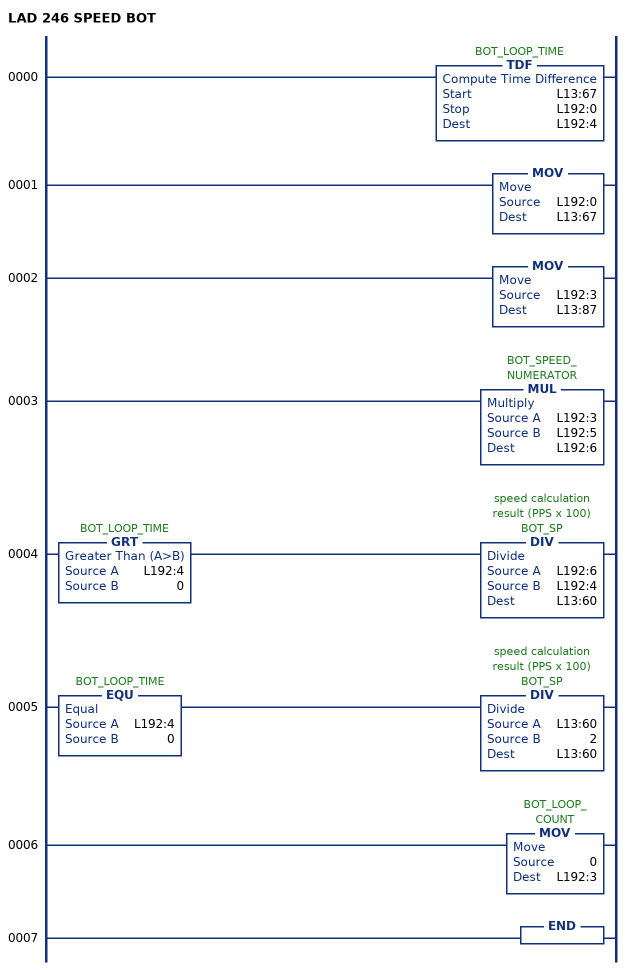
% Rung: 0 %
SOR TDF L13:67 L192:0 L192:4 EOR
%   L192:0  BOT_THIS_TIME  "rtc bot belt movement event time" %
%   L192:4  BOT_LOOP_TIME %
% Rung: 1 %
SOR MOV L192:0 L13:67 EOR
%   L192:0  BOT_THIS_TIME  "rtc bot belt movement event time" %
% Rung: 2 %
SOR MOV L192:3 L13:87 EOR
%   L192:3  BOT_LOOP_COUNT %
% Rung: 3 %
SOR MUL L192:3 L192:5 L192:6 EOR
%   L192:3  BOT_LOOP_COUNT %
%   L192:5  TKS_PER_SECOND %
%   L192:6  BOT_SPEED_NUMERATOR %
% Rung: 4 %
SOR GRT L192:4 0 DIV L192:6 L192:4 L13:60 EOR
%   L192:4  BOT_LOOP_TIME %
%   L192:6  BOT_SPEED_NUMERATOR %
%   L13:60  BOT_SP  "speed calculation result (PPS x 100)" %
% Rung: 5 %
SOR EQU L192:4 0 DIV L13:60 2 L13:60 EOR
%   L192:4  BOT_LOOP_TIME %
%   L13:60  BOT_SP  "speed calculation result (PPS x 100)" %
% Rung: 6 %
SOR MOV 0 L192:3 EOR
%   L192:3  BOT_LOOP_COUNT %
% Rung: 7 %
SOR END EOR

LADDER 248 "SPEED TOP"    % high speed %
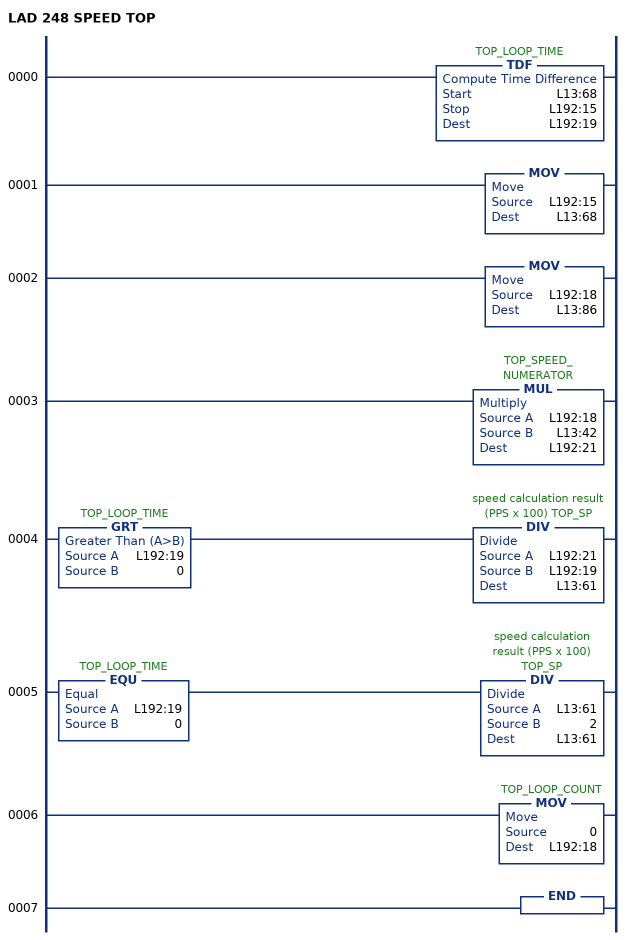
% Rung: 0 %
SOR TDF L13:68 L192:15 L192:19 EOR
%   L192:15  TOP_THIS_TIME  "rtc top belt movement event time" %
%   L192:19  TOP_LOOP_TIME %
% Rung: 1 %
SOR MOV L192:15 L13:68 EOR
%   L192:15  TOP_THIS_TIME  "rtc top belt movement event time" %
% Rung: 2 %
SOR MOV L192:18 L13:86 EOR
%   L192:18  TOP_LOOP_COUNT %
% Rung: 3 %
SOR MUL L192:18 L13:42 L192:21 EOR
%   L192:18  TOP_LOOP_COUNT %
%   L192:21  TOP_SPEED_NUMERATOR %
% Rung: 4 %
SOR GRT L192:19 0 DIV L192:21 L192:19 L13:61 EOR
%   L192:19  TOP_LOOP_TIME %
%   L192:21  TOP_SPEED_NUMERATOR %
%   L13:61  TOP_SP  "speed calculation result (PPS x 100)" %
% Rung: 5 %
SOR EQU L192:19 0 DIV L13:61 2 L13:61 EOR
%   L192:19  TOP_LOOP_TIME %
%   L13:61  TOP_SP  "speed calculation result (PPS x 100)" %
% Rung: 6 %
SOR MOV 0 L192:18 EOR
%   L192:18  TOP_LOOP_COUNT %
% Rung: 7 %
SOR END EOR

LADDER 250 "P BOT"    % high speed %
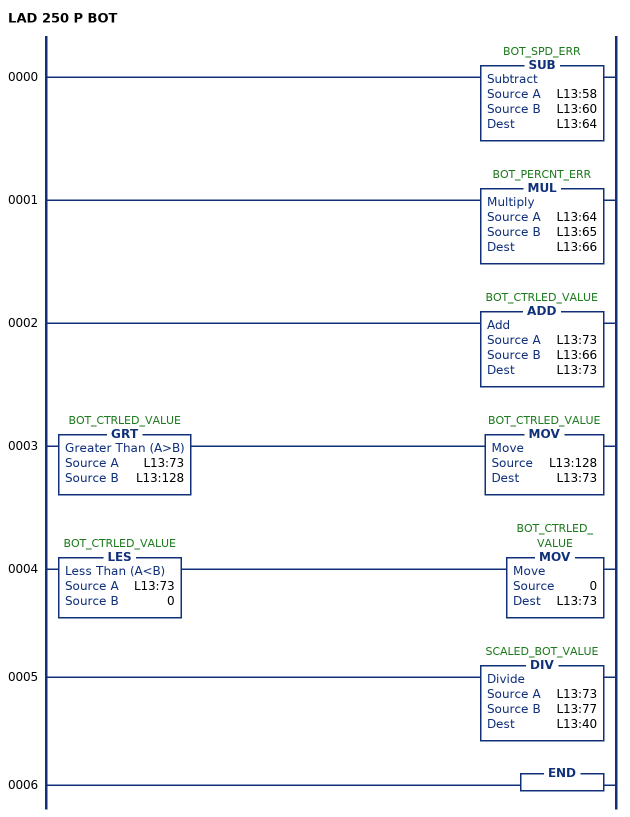
% Rung: 0 %
SOR SUB L13:58 L13:60 L13:64 EOR
%   L13:58  BOT_SPD_SETPOINT %
%   L13:60  BOT_SP  "speed calculation result (PPS x 100)" %
%   L13:64  BOT_SPD_ERR %
% Rung: 1 %
SOR MUL L13:64 L13:65 L13:66 EOR
%   L13:64  BOT_SPD_ERR %
%   L13:65  POS5SHIFT %
%   L13:66  BOT_PERCNT_ERR %
% Rung: 2 %
SOR ADD L13:73 L13:66 L13:73 EOR
%   L13:73  BOT_CTRLED_VALUE %
%   L13:66  BOT_PERCNT_ERR %
% Rung: 3 %
SOR GRT L13:73 L13:128 MOV L13:128 L13:73 EOR
%   L13:73  BOT_CTRLED_VALUE %
%   L13:128  "how much top has shifted since measurment" %
% Rung: 4 %
SOR LES L13:73 0 MOV 0 L13:73 EOR
%   L13:73  BOT_CTRLED_VALUE %
% Rung: 5 %
SOR DIV L13:73 L13:77 L13:40 EOR
%   L13:73  BOT_CTRLED_VALUE %
%   L13:40  SCALED_BOT_VALUE %
% Rung: 6 %
SOR END EOR

LADDER 252 "P TOP"    % high speed %
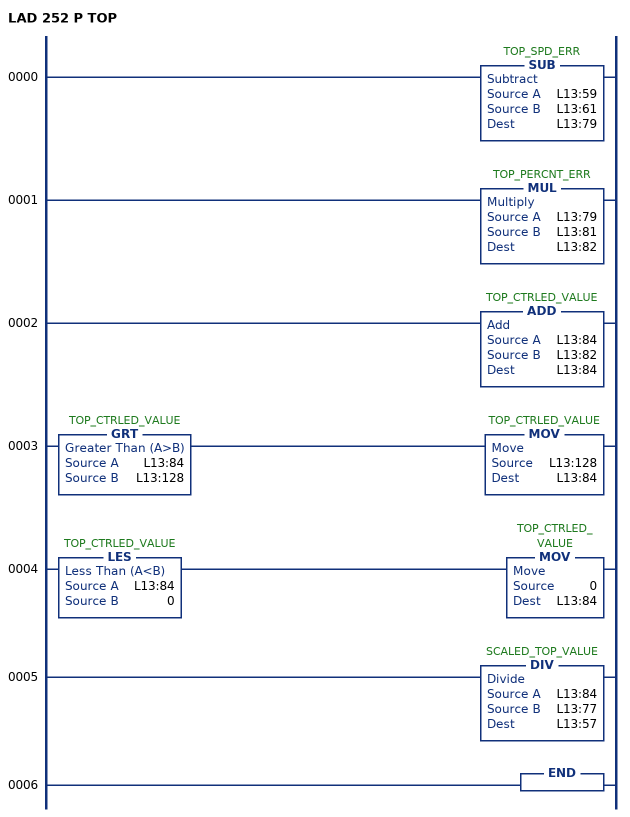
% Rung: 0 %
SOR SUB L13:59 L13:61 L13:79 EOR
%   L13:59  TOP_SPD_SETPOINT %
%   L13:61  TOP_SP  "speed calculation result (PPS x 100)" %
%   L13:79  TOP_SPD_ERR %
% Rung: 1 %
SOR MUL L13:79 L13:81 L13:82 EOR
%   L13:79  TOP_SPD_ERR %
%   L13:81  TOP_FDBK_RATIO %
%   L13:82  TOP_PERCNT_ERR %
% Rung: 2 %
SOR ADD L13:84 L13:82 L13:84 EOR
%   L13:84  TOP_CTRLED_VALUE %
%   L13:82  TOP_PERCNT_ERR %
% Rung: 3 %
SOR GRT L13:84 L13:128 MOV L13:128 L13:84 EOR
%   L13:84  TOP_CTRLED_VALUE %
%   L13:128  "how much top has shifted since measurment" %
% Rung: 4 %
SOR LES L13:84 0 MOV 0 L13:84 EOR
%   L13:84  TOP_CTRLED_VALUE %
% Rung: 5 %
SOR DIV L13:84 L13:77 L13:57 EOR
%   L13:84  TOP_CTRLED_VALUE %
%   L13:57  SCALED_TOP_VALUE %
% Rung: 6 %
SOR END EOR

LADDER 254 "TOTALCOUNT"
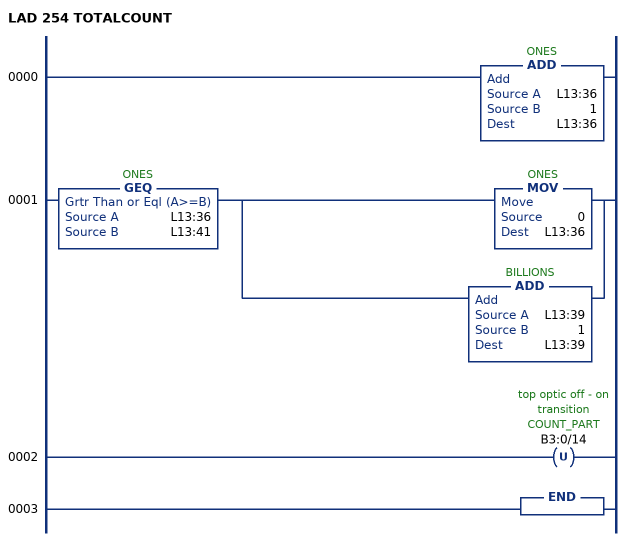
% Rung: 0 %
SOR ADD L13:36 1 L13:36 EOR
%   L13:36  ONES %
% Rung: 1 %
SOR GEQ L13:36 L13:41 BST MOV 0 L13:36 NXB ADD L13:39 1 L13:39 BND EOR
%   L13:36  ONES %
%   L13:41  "skipped count change in the last 3 seconds" %
%   L13:39  BILLIONS %
% Rung: 2 %
SOR OTU B3:0/14 EOR
%   B3:0/14  COUNT_PART  "top optic off - on transition" %
% Rung: 3 %
SOR END EOR

LADDER 255 "SAVED"
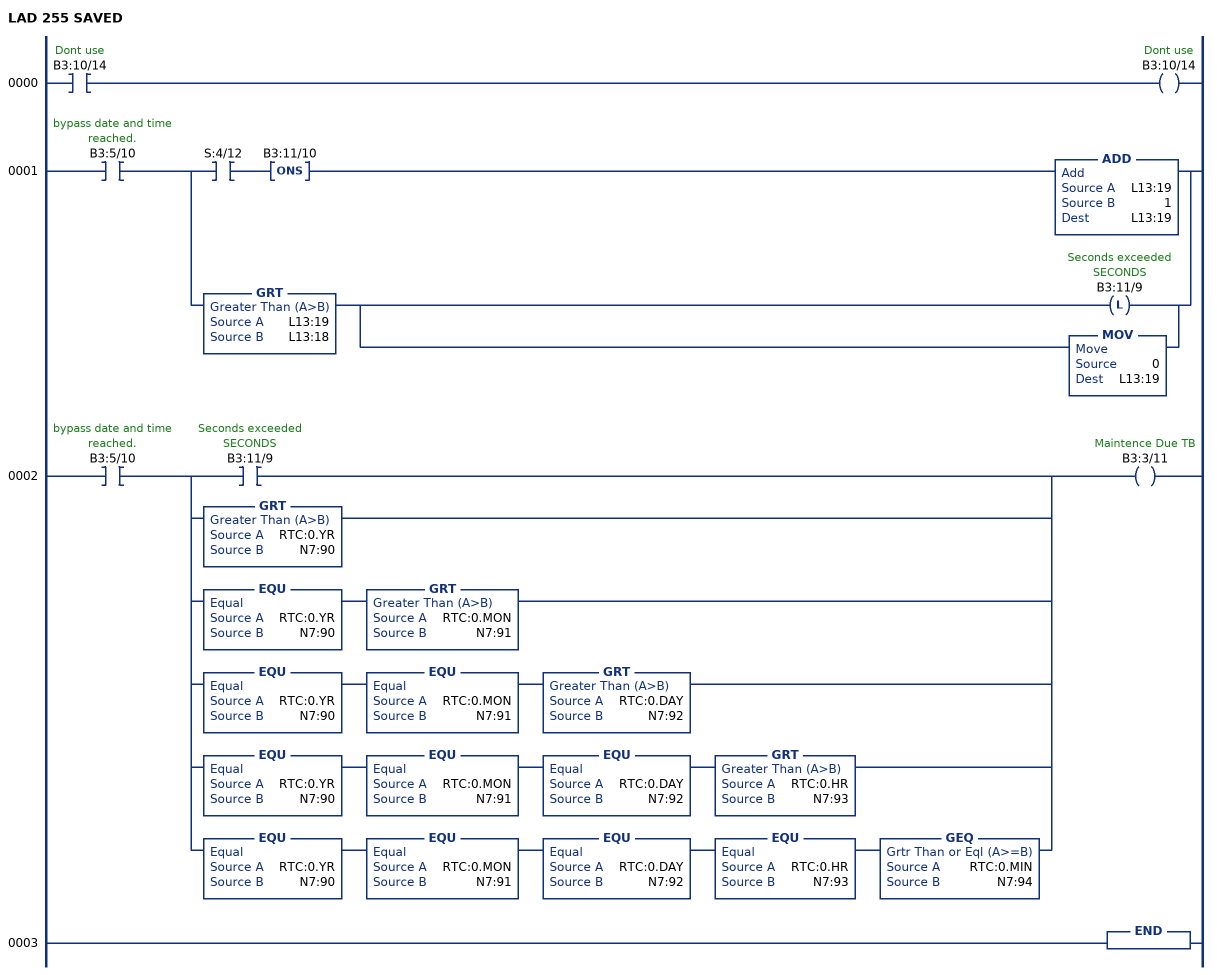
% Rung: 0 %
SOR XIC B3:10/14 OTE B3:10/14 EOR
%   B3:10/14  "Dont use" %
% Rung: 1 %
SOR XIC B3:5/10 BST XIC S:4/12 ONS B3:11/10 ADD L13:19 1 L13:19 NXB GRT L13:19 L13:18 BST OTL B3:11/9 NXB MOV 0 L13:19 BND BND EOR
%   B3:5/10  "bypass date and time reached." %
%   L13:18  MAX %
%   B3:11/9  SECONDS  "Seconds exceeded" %
% Rung: 2 %
SOR XIC B3:5/10 BST XIC B3:11/9 NXB GRT RTC:0.YR N7:90 NXB EQU RTC:0.YR N7:90 GRT RTC:0.MON N7:91 NXB EQU RTC:0.YR N7:90 EQU RTC:0.MON N7:91 GRT RTC:0.DAY N7:92 NXB EQU RTC:0.YR N7:90 EQU RTC:0.MON N7:91 EQU RTC:0.DAY N7:92 GRT RTC:0.HR N7:93 NXB EQU RTC:0.YR N7:90 EQU RTC:0.MON N7:91 EQU RTC:0.DAY N7:92 EQU RTC:0.HR N7:93 GEQ RTC:0.MIN N7:94 BND OTE B3:3/11 EOR
%   B3:5/10  "bypass date and time reached." %
%   B3:11/9  SECONDS  "Seconds exceeded" %
%   N7:90  RTC %
%   B3:3/11  TB  "Maintence Due" %
% Rung: 3 %
SOR END EOR

OTHER DOCUMENTED ADDRESSES
  B189:0/0  "change box"
  B189:0/9  "override boxing ok or not full signal"
  B189:0/11  "HMI force door close"
  B196:1/0  "Chute door is closed"
  B196:1/1  "control chute door"
  B196:1/13  "force box conveyor on"
  B196:3/0  "for hmi to continue production unlatched by hmi"
  HSC:0.0  "top"
  HSC:0.3/6  "Underflow interrupt"
  HSC:0.3/7  "Overflow interrupt"
  HSC:1.0  "bot"
  HSC:1.3/6  "Underflow interrupt"
  HSC:1.3/7  "Overflow interrupt"
  I:0.0/0  "Encoder Signal "A""
  I:0.0/1  "Encoder Signal "B""
  I:0.0/4  "Encoder Signal "A""
  I:0.0/5  "Encoder Signal "B""
  I:0.1/4  "not used"
  I:0.1/5  "not used"
  I:0.1/6  "not used"
  I:0.1/7  "not used"
  I:0.1/8  "not used"
  I:0.1/9  "not used"
  I:0.1/10  "not used"
  I:0.1/11  "not used"
  I:0.1/12  "not used"
  I:0.1/13  "not used"
  I:0.1/14  "not used"
  I:0.1/15  "not used"
  I:0.2  "not used"
  I:0.2/3  "Packaging Conveyor full"
  I:0.2/4  "Packaging Conveyor Box in Position"
  I:0.3  "not used"
  I:0.4  "Spare Analog Input 1"
  I:0.5  "Spare Analog Input 2"
  I:0.6  "Spare Analog Input 3"
  I:2.0/0  FRONT_ESTOP
  I:2.0/1  REAR_ESTOP
  I:2.0/8  FRONT_DOOR  "front door signal ce models only"
  I:2.0/9  REAR_DOOR  "rear door signal ce models only"
  I:2.0/11  "spare"
  I:2.0/12  "spare"
  I:2.0/14  "spare"
  L13:180  "maximum time between triggers"
  L13:181  "minimum okay time between triggers"
  L13:182  RATE_QUEUE_LIMIT
  L13:184  "intermediate i1 trig avg"
  L13:185  I1_TBT  "i1 average time between triggers"
  L13:186  "intermediate i5 trig avg"
  L13:187  I5_TBT  "i5 average time between triggers"
  L13:188  "intermediate i6 trig avg"
  L13:189  I6_TBT  "i6 average time between triggers"
  L13:190  "i1 timed q limit"
  L13:191  "i1 absolute q limit"
  L16:2  TRIG_DELAY_Q_MULTI
  L16:3  TRIG_DELAY_MIN_TIME
  L16:4  TRIG_DELAY_FLAT_RATE
  L16:5  CLEARTIME1  "time to clear tracking data"
  L16:6  CLEARTIME5
  L16:7  CLEARTIME6
  L16:8  PASS1PRTLOC
  L16:9  PASS1PROCESSTM
  L16:11  PASS5PROCESSTM
  L16:13  PASS6PROCESSTM
  L23:19  TOP_OPT_FAIL_CT
  L23:34  AIR_PRESSURE_FAULT
  L28:0  INS_1_TIME
  L29:0  INS_1_POS
  L30:0  INS_5_TIME
  L31:0  INS_5_POS
  L32:0  INS_6_TIME
  L33:0  INS_6_POS
  L192:1  BOT_LAST_TIME  "rtc bot belt previous movement event time"
  L192:2  BOT_CYCLE_TIME  "rtc bot belt time between events"
  L192:7  FROM_REAL  "distance from real part signal at optic location"
  L192:8  FROM_TRACKED  "distance from tracked part signal at optic location"
  L192:16  TOP_LAST_TIME  "rtc top belt previous movement event time"
  L192:17  TOP_CYCLE_TIME  "rtc top belt time between events"
  L199:5  ACQTM51
  L199:6  ACQTM52
  L199:7  ACQTM53
  L199:9  "ones"
  L199:10  "billions"
  L199:13  DUMP_LONG
  L199:15  ACQTM11
  L199:16  ACQTM12
  L199:17  ACQTM13
  L199:20  RESULTTM1
  L199:22  CLEARTIME5COUNT
  L199:23  CLEARTIME6COUNT
  L199:24  ACQTM61
  L199:25  ACQTM62
  L199:26  ACQTM63
  L199:27  TMSINCETRIG1
  L199:29  TMSINCETRIG5
  L199:30  TMSINCETRIG6
  L199:31  CLEARTIME1COUNT
  L199:32  RESULTTM5
  L199:33  RESULTTM6
  L199:34  MAXACQTM1
  L199:36  MAXACQTM6
  N7:45  I5_MAX_SHIFT  "ins 5 maximum result location"
  N7:47  I6_MAX_SHIFT  "ins 6 maximum result location"
  N7:84  I7_MAX_SHIFT
  N7:85  I8_MAX_SHIFT
  N15:5  INS_1_TRIG_LOC
  O:0.0/1  "spare"
  O:0.0/5  INS_8_TRIG  "Inspection 8 Trigger"
  O:0.0/11  "Spare"
  O:0.0/12  "not used"
  O:0.0/13  "not used"
  O:0.0/14  "not used"
  O:0.0/15  "not used"
  O:0.1  "not used"
  O:0.2  "not used"
  O:0.3  "not used"
  O:0.5  "spare analog output"
  O:3.0/0  "spare"
  O:3.0/2  "spare"
  O:3.0/3  "light curtain range selection /* needed? */"
  O:3.0/7  "door unlocks on CE models"
  O:3.0/8  "spare"
  O:3.0/9  "spare"
  O:3.0/10  "spare"
  O:3.0/11  FEEDWHEEL
  PFILE:6  "check for part jams"
  PFILE:10  "Bottom belt HSC"
  PFILE:12  "Top belt HSC"
  Q2:55  END_OF_MAIN
  Q5:94  END_OF_BELTS
  T20:0  "Trigger On Time"
  U:9  "slow data"
  U:11  "transfered data calcuations from the high speed section"
  U:24  "check skipped fail rate"
  U:28  "faults"
  U:29  "speed"
  U:30  "count"
  U:31  "rate calc"
  U:32  "boxer"
  U:33  "bulk pack"
  U:34  "customer boxing unit signals"
  U:35  "cleanup"
  U:180  "rate calc"

COMMENTS NOT ATTACHED TO A CURRENT RUNG
  RUNG000150-000041: transfer tracked part positon from trigger/acquire to the acquire/result
    capture acquire time
    reset process time
  RUNG000150-000039: Grab trigger/acquire position
    Grab acquire time
  RUNG000150-000038: acquire code
  RUNG000150-000035: fail count
  RUNG000150-000032: pass count
  RUNG000150-000025: pass code / Set pass bit in Bit Shift
    captures result position and processing time
    Unlatch pass bit
  RUNG000150-000018: pass, fail and acquire inputs
  RUNG000150-000016: wiped count
  RUNG000150-000014: clear data for time
  RUNG000150-000013: clear data for aquire time expired
  RUNG000150-000012: wipe stored part data if acq time expires
  RUNG000150-000011: trigger count
  RUNG000010-000018: Remove any part present signals outside of expected location
  RUNG000010-000014: ****
                      Zeros out the non passing part count when one passes
    ****
  RUNG000125-000011: trigger count
  RUNG000125-000012: wipe stored part data if acq time expires
  RUNG000125-000013: clear data for aquire time expired
  RUNG000125-000014: clear data for time
  RUNG000125-000016: wiped count
  RUNG000125-000018: pass, fail and acquire inputs
  RUNG000125-000025: pass code / Set pass bit in Bit Shift
    captures result position and processing time
    Unlatch pass bit
  RUNG000125-000026: Grab trigger/acquire position
    Grab acquire time
  RUNG000125-000027: transfer tracked part positon from trigger/acquire to the acquire/result
    capture acquire time
    reset process time
  RUNG000125-000029: Set pass bit in Bit Shift
    captures result position and processing time
    Unlatch pass bit

REVISION NOTES
  13: updated count reset
  14: added io moduals
  15: multiple steps toward new hmi integration
  21: test
  27: fix error if bulk pack and no boxing fallout were on

DATA TABLE (non-zero values as saved)
DATA B3
% B3:0 % 0XA020 0X0260 0X4000 0XA001 0XCEFF 0X5540 0X0024 0X0421 0X5F80 0X24D0
% B3:10 % 0X21E0 0X0006 0X2000 0X0000
DATA T4
% .PRE .ACC %
% T4:1 % 150 150
% T4:2 % 400 0
% T4:3 % 222 0
% T4:4 % 300 0
% T4:5 % 5 5
% T4:6 % 10 10
% T4:7 % 20000 20001
% T4:8 % 20 18
% T4:9 % 50 17
% T4:10 % 200 200
% T4:11 % 3000 1300
% T4:12 % 55 55
% T4:13 % 250 0
% T4:14 % 666 0
% T4:15 % 1000 1002
% T4:16 % 400 0
% T4:17 % 100 26
% T4:18 % 5 0
% T4:19 % 300 0
% T4:20 % 200 0
% T4:21 % 200 0
% T4:22 % 200 0
% T4:23 % 250 0
% T4:24 % 666 0
% T4:25 % 666 0
% T4:26 % 666 0
% T4:27 % 250 0
% T4:28 % 250 0
% T4:29 % 5000 0
% T4:30 % 222 48
% T4:31 % 222 49
% T4:32 % 222 51
% T4:33 % 222 34
DATA C5
% .PRE .ACC %
% C5:0 % 32766 0
DATA R6
% .LEN .POS %
% R6:0 % 1250 0
% R6:1 % 1250 0
% R6:2 % 1024 0
% R6:3 % 1024 0
% R6:4 % 1250 0
% R6:5 % 1250 0
% R6:6 % 1713 0
% R6:7 % 1024 0
% R6:8 % 1024 0
% R6:9 % 3 0
% R6:10 % 1713 0
% R6:11 % 1713 0
% R6:12 % 10 0
% R6:13 % 10 0
% R6:14 % 10 0
% R6:15 % 10 0
% R6:16 % 1713 0
% R6:17 % 1713 0
% R6:18 % 1713 0
% R6:19 % 10 0
DATA N7
% N7:0 % 32767 3 634 300 18 400 0 32767 500 500
% N7:10 % 1000 18 0 2 20 20 1000 2000 50 1050
% N7:20 % 32767 222 10 222 222 46 48 0 48 250
% N7:30 % 666 2023 150 0 0 1056 66 33 0 33
% N7:40 % 0 26 1 25 727 482 32767 632 2967 13
% N7:50 % 12 16 13 16 17 1024 17365 8191 32766 18
% N7:60 % 1713 1713 1713 1021 580 560 4999 5 400 400
% N7:70 % 100 200 300 400 90 190 290 390 9536 25486
% N7:80 % 0 0 1059 1075 832 844 42 44 0 0
% N7:90 % 2011 4 4 12 1 42 44 222 222 12
% N7:100 % 1003 90 110 100 175 25 0 0 0 0
DATA F8
% F8:0 % 6 1 23807 499 0.23807
% F8:5 % 0 0 500 1.9 2
% F8:10 % 1 0.08897486 3058 101 63.26563
% F8:15 % 37.73437 4040 2 0 0
% F8:20 % 0 0.02 0 1 0
% F8:25 % 0 932781 0.222 279.6551 848597
% F8:30 % 0 170 0.03 38 852060
% F8:35 % 0 0 0 0 77
% F8:40 % 101 37.73437 0 100 1
% F8:45 % 1 2 0.21455 0 0
% F8:50 % 0 0 1 0 1
% F8:55 % 2000000 -221 0 0 0
% F8:95 % 0 0 0 492 4.92
DATA B12
% B12:0 % 0X6144 0X0000 0X0000 0X0000 0X0000 0X0000 0X0000 0X0000 0X0000 0X0000
DATA L13
% L13:0 % 4145 42892 98977 24252 50258
% L13:5 % 0 17605 0 45196 672
% L13:10 % 15 18734415 10060 18 90
% L13:15 % 2111548362 -2147483648 2147483647 2147483647 82058
% L13:20 % 1326931947 1715820752 777 100 100
% L13:25 % 153441500 49 684 0 1784530491
% L13:30 % 327017240 19112 1020000 2110915449 444
% L13:35 % 0 96146 0 0 0
% L13:40 % 0 1000000000 1000000 2110915422 2109978324
% L13:45 % 2110917187 150 0 27 1715693141
% L13:50 % 1570077 632979 1185380638 0 0
% L13:55 % 631214 523785 9175 0 2000
% L13:60 % 0 2000 27 600 0
% L13:65 % 100 0 2044072 1569509921 -942969229
% L13:70 % 1612034666 772154329 64 0 1715693141
% L13:75 % 18 60 100 1182976851 0
% L13:80 % 772154329 50 0 1 917450
% L13:85 % 127698 102 0 0 5
% L13:90 % 10 5 96146 10 2109978349
% L13:95 % 10 937137 0 2110917215 203866
% L13:100 % 6400 0 2147483647 9460280 227
% L13:105 % 203866 772154618 1326019172 133426 1326019166
% L13:110 % 6 100 30 1696958651 1715692998
% L13:115 % 1715693066 68 34 1715693032 1
% L13:120 % 75232332 3889 30 100 23
% L13:125 % 0 1612034666 2147483647 3276500 18862123
% L13:130 % 2 2 0 99 0
% L13:135 % 0 0 127708 5 0
% L13:140 % 1 5 36 50 50
% L13:145 % 5 5 5 5 4
% L13:150 % 15 25 46 -46 18734415
% L13:155 % 0 -9 0 0 4589052
% L13:160 % 10 25 28 25 28
% L13:165 % 1715616164 1715693497 1715616164 1715693497 47547
% L13:170 % 127144 225 938827 1000 2300
% L13:175 % 4 0 42 23 38
% L13:180 % 176247033 25 99000 52866 644409
% L13:185 % 64 916459 92 627156 63
% L13:190 % 4 5 0 0 0
DATA F14
% F14:0 % 1.32889e-38 5747.126 1550 1550 1638.3
% F14:5 % 1638.3 1638.3 1638.3 0 0
DATA N15
% N15:0 % 1055 1065 1275 900 709 105 66 1186 600 10
% N15:10 % 71 887 0 0 0 0 1356 0 0 0
DATA L16
% L16:0 % 16 55 11 0 20
% L16:5 % 250 5000 5000 182 19
% L16:10 % 1256 18 2045 6599584 98
% L16:15 % 99 0 0 0 0
DATA L19
% L19:0 % 1786464927 1786485574 1786536494 1786569665 1789039725
% L19:5 % 1789053785 1789107296 1789133049 1789181522 1789191558
% L19:10 % 1789214193 1789244752 2110915051 1784530491 1784545122
% L19:15 % 1784592142 1786431837 0 0 0
DATA L20
% L20:0 % 2051345556 2051345781 2051346006 2109372928 2109373154
% L20:5 % 2109373380 2109373607 2109373832 2109374060 2109374287
% L20:10 % 2109374512 2109374739 2109374964 2109438205 2109438431
% L20:15 % 2109438657 2109438883 2109439109 2109439335 2109439560
% L20:20 % 2109439787 2109440013 2109440238 2109676669 2109676896
% L20:25 % 2109677122 2109677349 2109677576 2109677802 2109678029
% L20:30 % 2109678254 2109678480 2109678708 2109976290 2109976516
% L20:35 % 2109976742 2109976968 2109977194 2109977420 2109977646
% L20:40 % 2109977873 2109978099 2109978324 2051343975 2051344201
% L20:45 % 2051344426 2051344652 2051344878 2051345104 2051345330
DATA L21
% L21:0 % 1701145872 1701145874 1701145876 1715554020 1715554061
% L21:5 % 1715554099 1715554135 1715554168 1715554200 1715554229
% L21:10 % 1715554256 1715554281 1715554304 1715555145 1715555147
% L21:15 % 1715555150 1715555152 1715555154 1715555156 1715555158
% L21:20 % 1715555161 1715555163 1715555166 1715583713 1715583754
% L21:25 % 1715583793 1715583830 1715583864 1715583896 1715583926
% L21:30 % 1715583953 1715583978 1715584002 1715615849 1715615892
% L21:35 % 1715615934 1715615974 1715616011 1715616046 1715616079
% L21:40 % 1715616110 1715616138 1715616164 1701145856 1701145858
% L21:45 % 1701145860 1701145862 1701145865 1701145867 1701145869
DATA L22
% L22:0 % 1788993602 1789041980 1789056046 1789109557 1789135315
% L22:5 % 1789183783 1789193818 1789216454 1789247013 1789550452
% L22:10 % 1789550678 1789552037 1789552263 1789552490 1792306301
% L22:15 % 1792306527 1792307883 1792308111 1792308338 2051343994
% L22:20 % 2051344219 2051345571 2051345796 2051346023 2109372945
% L22:25 % 2109373172 2109374528 2109374755 2109374982 2109438224
% L22:30 % 2109438449 2109439805 2109440031 2109440257 2109676687
% L22:35 % 2109676915 2109678271 2109678497 2109678722 2109976321
% L22:40 % 2109976547 2109977907 2109978134 2109978360 2110917187
% L22:45 % 1788992473 1788992698 1788992925 1788993150 1788993376
DATA L23
% L23:0 % 1697873055 1697874460 1697877298 1697888087 1697893281
% L23:5 % 1697903053 1697905076 1697909640 1697915801 1697976977
% L23:10 % 1697977022 1697977296 1697977342 1697977387 1698532583
% L23:15 % 1698532629 1698532903 1698532949 1698532994 1701145856
% L23:20 % 1701145858 1701145872 1701145874 1701145876 1715554023
% L23:25 % 1715554064 1715554258 1715554282 1715554305 1715555145
% L23:30 % 1715555147 1715555161 1715555163 1715555166 1715583716
% L23:35 % 1715583758 1715583955 1715583980 1715584003 1715615855
% L23:40 % 1715615898 1715616114 1715616142 1715616168 1715693497
% L23:45 % 1697873055 1697873055 1697873055 1697873055 1697873055
DATA L30
% L30:0 % 1789551973 1789552201 1789552428 1792306242 1792306468
% L30:5 % 1792307826 1792308054 1792308280 2051343935 2051344160
% L30:10 % 2051345518 2051345744 2051345971 2109372887 2109373113
% L30:15 % 2109374471 2109374698 2109374922 2109438166 2109438391
% L30:20 % 2109439748 2109439975 2109440201 2109676630 2109676856
% L30:25 % 2109678214 2109678440 2109678666 2109976249 2109976475
% L30:30 % 2109977832 2109978060 2109978285 2110915422 1786570159
% L30:35 % 1788738453 1788738679 1788740036 1788740261 1788740487
% L30:40 % 1789040217 1789054280 1789107790 1789133548 1789182016
% L30:45 % 1789192054 1789214689 1789245248 1789550391 1789550617
DATA L31
% L31:0 % 1697977283 1697977329 1697977375 1698532571 1698532617
% L31:5 % 1698532891 1698532937 1698532982 1701145855 1701145857
% L31:10 % 1701145871 1701145874 1701145876 1715554012 1715554053
% L31:15 % 1715554251 1715554276 1715554299 1715555145 1715555147
% L31:20 % 1715555161 1715555163 1715555165 1715583706 1715583747
% L31:25 % 1715583948 1715583974 1715583998 1715615840 1715615884
% L31:30 % 1715616105 1715616133 1715616160 1715693141 1697530761
% L31:35 % 1697873055 1697873055 1697873055 1697873055 1697873055
% L31:40 % 1697874104 1697876942 1697887731 1697892925 1697902697
% L31:45 % 1697904720 1697909284 1697915445 1697976964 1697977010
DATA L32
% L32:0 % 1185360253 1185361609 1185361836 1185363193 1185363419
% L32:5 % 1185364779 1185365005 1185366360 1185366586 1185367942
% L32:10 % 1185368169 1185369529 1185369756 1185371117 1185371345
% L32:15 % 1185372706 1185372932 1185374289 1185374515 1185375875
% L32:20 % 1185376102 1185377462 1185377689 1185379050 1185379278
% L32:25 % 1185380638 1185380865 1185342586 1185342813 1185344174
% L32:30 % 1185344401 1185345759 1185345985 1185347343 1185347569
% L32:35 % 1185348928 1185349154 1185350512 1185350739 1185352100
% L32:40 % 1185352326 1185353684 1185353910 1185355270 1185355497
% L32:45 % 1185356855 1185357081 1185358440 1185358666 1185360026
DATA L33
% L33:0 % 1687266998 1687266998 1687266998 1687266998 1687266998
% L33:5 % 1687266998 1687266998 1687266998 1687266998 1687266998
% L33:10 % 1687266998 1687266998 1687266998 1687266998 1687266998
% L33:15 % 1687266998 1687266998 1687266998 1687266998 1687266998
% L33:20 % 1687266998 1687266998 1687266998 1687266998 1687266998
% L33:25 % 1687266998 1687266998 1687266998 1687266998 1687266998
% L33:30 % 1687266998 1687266998 1687266998 1687266998 1687266998
% L33:35 % 1687266998 1687266998 1687266998 1687266998 1687266998
% L33:40 % 1687266998 1687266998 1687266998 1687266998 1687266998
% L33:45 % 1687266998 1687266998 1687266998 1687266998 1687266998
DATA B37
% B37:0 % 0X0000 0X0000 0X0000 0X0000 0X0000 0X0000 0X0000 0X0002 0X0000 0X0000
DATA B38
% B38:0 % 0X0000 0X0000 0X0000 0X0000 0X0000 0X0000 0X0000 0X0002 0X0000 0X0000
% B38:10 % 0X0000 0X0000 0X0000 0X0000 0X0000 0X0000 0X0000 0X0000 0XE000 0XFFFE
% B38:20 % 0X007C 0X2000 0X0000 0X0000 0X0000 0X0000 0X0000 0X0000 0X0000 0X0000
% B38:30 % 0X0000 0X0000 0X0000 0X0000 0X0000 0X0000 0X0000 0X6000 0X0007 0X0400
% B38:40 % 0X0000 0X0000 0X0000 0X0000 0X0040 0X8800 0X0080 0X0000 0X0000 0X0000
% B38:50 % 0X2000 0X0000 0X0000 0X0000 0X0000 0X0000 0X0000 0X0000 0X0000 0X0000
% B38:60 % 0X8000 0X0810 0X0000 0X8800 0X0003 0X0000 0X0FFF 0X0000 0X0000 0X0000
% B38:120 % 0X0000 0X0000 0X0000 0X0000 0X0000 0X0000 0X0000 0X0002
DATA B39
% B39:0 % 0X0000 0X0000 0X0000 0X0000 0X0000 0X0000 0X0000 0X0002 0X0000 0X0000
DATA B40
% B40:0 % 0X0000 0X0000 0X0000 0X0000 0X0000 0X0000 0X0000 0X0002 0X0000 0X0000
% B40:10 % 0X0000 0X0000 0X0000 0X0000 0X0000 0X0000 0X0000 0X0000 0XE000 0XFFFE
% B40:20 % 0X007C 0X2000 0X0000 0X0000 0X0000 0X0000 0X0000 0X0000 0X0000 0X0000
% B40:30 % 0X0000 0X0000 0X0000 0X0000 0X0000 0X0000 0X0000 0X6000 0X0007 0X0400
% B40:40 % 0X0000 0X0000 0X0000 0X0000 0X0040 0X8800 0X0080 0X0000 0X0000 0X0000
% B40:50 % 0X2000 0X0000 0X0000 0X0000 0X0000 0X0000 0X0000 0X0000 0X0000 0X0000
% B40:60 % 0X8000 0X0810 0X0000 0X8800 0X0003 0X0000 0X0FFF 0X0000 0X0000 0X0000
% B40:120 % 0X0000 0X0000 0X0000 0X0000 0X0000 0X0000 0X0000 0X0002
DATA L192
% L192:0 % 2044072 266932201 5055 0 0
% L192:5 % 1000000 0 999 999 8
% L192:10 % 0 0 0 78 17
% L192:15 % 1569679044 332250347 860888 33 50983
% L192:20 % 180 102000000 0 0 0
DATA B196
% B196:0 % 0X0A24 0X9FF2 0X0005 0X0000 0X0000 0X0000 0X0000 0X0000 0X0000 0X0000
% B196:30 % 0XE800 0X9BFF 0XEBFF 0XFFDF 0XFFFF 0X0000 0X0000 0X0000 0X0000 0X0000
DATA L199
% L199:0 % 1 0 0 0 0
